{attribute 'qualified_only'}
{attribute 'strict'}
{attribute 'to_string'}
TYPE BottomMaterialsEnum :
(

	//CARDBOARD
	CAR20S, CAR20M, CAR20L, CAR28S, CAR28M, CAR28L, //base (flat)
	
	//CHIPBOARD
	CIP18, CIP54,
	
	//WOOD BUNK
	WDB20, WDB22, WDB28, //bottom
	
	size //number of materials
);
END_TYPE

(* stored: Version 1.1.0.1, ProductVersion 3.1.4024.11
   EnumerationTextList BottomMaterialsEnum: Id {c93dc77b-1cac-46bc-ba0e-6184c6a1b5b7} *)
